//EL5021 | 1-channel Sin/Cos encoder
FUNCTION_BLOCK EL5021

VAR_INPUT
    En              : BOOL;
    iTerminal_ID    : INT;
    ErrorSystem     : POINTER TO ST_ErrorSystem;
END_VAR

VAR_OUTPUT
    EnO     : BOOL;
    bError  : BOOL;
	sErrorMessage: STRING;
END_VAR

VAR
    
    InfoData_State      AT %I*  : UINT;
    WcState_WcState     AT %I*  : BOOL;
    
    //FB-s
    EL5021_Error    : FB_TerminalError;
	
END_VAR

(*
* TODO: Test on hardware
*)
EnO:=En;

//Error FB instances
EL5021_Error(
    En                  := TRUE,
    iTerminal_ID        := iTerminal_ID,
    bWcState            := WcState_WcState,
    uiInfoData_State    := InfoData_State,
    pErrorSystem        := ErrorSystem,
    bError => bError,
);

IF bError THEN
    sErrorMessage:=EL5021_Error.ErrorData.sErrorMessage;
ELSE
	sErrorMessage:='';
END_IF

END_FUNCTION_BLOCK

(* stored: Version 1.1.0.1, ProductVersion 3.1.4024.6
   POU EL5021: Id {7f517c2d-3257-42d3-9c58-98a243359439}, SpecialFunc None *)
